FUNCTION_BLOCK FB_Depalletizer_1 IMPLEMENTS ITF_Depalletizer
VAR_INPUT
	Schuif : ITF_MotorSchuif;
	Zuignap1 : ITF_Vacuumzuignap;
	Zuignap2 : ITF_Vacuumzuignap;
	Zuignap3 : ITF_Vacuumzuignap;
	Zuignap4 : ITF_Vacuumzuignap;
	Druksensor1 : ITF_Druksensor;
	KlepDepallet : ITF_UnitKlep;

END_VAR
VAR_OUTPUT
END_VAR
VAR
	InputStateDep : E_PackMLStates;	
	CurrentStateDep : E_PackMLStates;



	testbool : BOOL;
	testbool2 : BOOL;
	GelezenStatusMotorSchuif : E_MotorSchuifStatus;
	GelezenStatusVacuumzuignap : E_VacuumzuignapStatus;
	GelezenDruk : REAL;
	GelezenStatusDruksensor : E_DruksensorStatus;
END_VAR

CASE InputStateDep OF

    E_PackMLStates.Idle:
        Idle();

    E_PackMLStates.Starting:
        Starting();

    E_PackMLStates.Execute:
        Execute();

    E_PackMLStates.Resetting:
        Resetting();

    E_PackMLStates.Holding:
        Holding();

    E_PackMLStates.Held:
        Held();

    E_PackMLStates.Unholding:
        Unholding();

    E_PackMLStates.Suspending:
        Suspending();

    E_PackMLStates.Suspended:
        Suspended();

    E_PackMLStates.Unsuspending:
        Unsuspending();

    E_PackMLStates.Stopping:
        Stopping();

    E_PackMLStates.Stopped:
        Stopped();

    E_PackMLStates.Aborting:
        Aborting();

    E_PackMLStates.Aborted:
        Aborted();

    E_PackMLStates.Clearing:
        Clearing();

END_CASE


















IF testbool = TRUE THEN
	Schuif.SturingKort();
	Zuignap1.Loslaten();
END_IF

IF testbool2 = TRUE THEN
	Schuif.SturingLang();
	Zuignap1.Oppakken();
END_IF

GelezenStatusMotorSchuif := Schuif.Status;
GelezenStatusVacuumzuignap := Zuignap1.Status;
GelezenDruk := Druksensor1.Druk;
GelezenStatusDruksensor := Druksensor1.Status;

METHOD Aborted : BOOL
VAR_INPUT
END_VAR
END_METHOD

METHOD Aborting : BOOL
VAR_INPUT
END_VAR
END_METHOD

METHOD Clearing : BOOL
VAR_INPUT
END_VAR
END_METHOD

PROPERTY CurrentState : E_PackMLStates
GET
CurrentState := CurrentStateDep;
END_GET
SET
CurrentStateDep := CurrentState;
END_SET
END_PROPERTY

METHOD Execute : BOOL
VAR_INPUT
END_VAR
END_METHOD

METHOD Held : BOOL
VAR_INPUT
END_VAR
END_METHOD

METHOD Holding : BOOL
VAR_INPUT
END_VAR
END_METHOD

METHOD Idle : BOOL
VAR_INPUT
END_VAR
CurrentStateDep := E_PackMLStates.Idle;
END_METHOD

PROPERTY InputState : E_PackMLStates
GET
InputState := InputStateDep;
END_GET
SET
InputStateDep := InputState;
END_SET
END_PROPERTY

METHOD Resetting : BOOL
VAR_INPUT
END_VAR
END_METHOD

METHOD Starting : BOOL
VAR_INPUT
END_VAR
CurrentStateDep := E_PackMLStates.Starting;

IF  Schuif.Status = E_MotorSchuifStatus.Kort AND Zuignap1.Status = E_VacuumzuignapStatus.SturingVacuumLoslaten AND
	Zuignap2.Status = E_VacuumzuignapStatus.SturingVacuumLoslaten AND Zuignap3.Status = E_VacuumzuignapStatus.SturingVacuumLoslaten AND
	Zuignap4.Status = E_VacuumzuignapStatus.SturingVacuumLoslaten AND DrukSensor1.Status = E_DruksensorStatus.SensorInputOk AND 
	KlepDepallet.Status = FALSE  THEN //vergeet de andere voorwaarden niet !!!!!
	
	CurrentStateDep := E_PackMLStates.Idle;
	ELSE
		Schuif.SturingKort();
		Zuignap1.Loslaten();
		Zuignap2.Loslaten();
		Zuignap3.Loslaten();
		Zuignap4.Loslaten();
		KlepDepallet.SturingOpen(FALSE); 
END_IF
END_METHOD

METHOD Stopped : BOOL
VAR_INPUT
END_VAR
END_METHOD

METHOD Stopping : BOOL
VAR_INPUT
END_VAR
END_METHOD

METHOD Suspended : BOOL
VAR_INPUT
END_VAR
END_METHOD

METHOD Suspending : BOOL
VAR_INPUT
END_VAR
END_METHOD

METHOD Unholding : BOOL
VAR_INPUT
END_VAR
END_METHOD

METHOD Unsuspending : BOOL
VAR_INPUT
END_VAR
END_METHOD

END_FUNCTION_BLOCK

(* stored: Version 1.1.0.1
   POU FB_Depalletizer_1: Id {604c825a-b299-42a4-9d94-06f2cd7a73fd}, SpecialFunc None
   Folder Methods: Id {41eb30da-c817-4a57-90b2-9b373696aeab}
   Folder Properties: Id {0a932fc3-77da-47ab-9595-fa212dce3ce7}
   Method Aborted: Id {0bfc1c67-cbbf-4ee0-9411-dfa1daf9e1fa}
   Method Aborting: Id {874fcde3-a461-43b7-8542-2e8c8f07c54a}
   Method Clearing: Id {a7e21cb3-b81b-4227-8a32-6a19ec30fdab}
   Property CurrentState: Id {5521c871-13ed-4e4c-a9b3-60eda6f215d2}
   Get Get: Id {abf65026-5da4-4773-9ad7-0771ec9a23a9}
   Set Set: Id {6aece2b5-c6a5-460d-8bf7-a59f80b5ecaa}
   Method Execute: Id {7bc828e8-56fb-4ceb-956d-11c06042b4fa}
   Method Held: Id {abf5bffe-4e53-4e4f-a0f2-17eb456b0638}
   Method Holding: Id {9ee0f93f-9ee6-40ae-91af-7b218154d752}
   Method Idle: Id {53c5baf1-bd08-4e97-999e-1b6af5cbd2b8}
   Property InputState: Id {4302f528-8764-4bef-8b72-acc9ee6f8e24}
   Get Get: Id {e211b0f1-ab3b-4059-8fd8-0ad7c175cd84}
   Set Set: Id {9bfc232a-27d2-4dce-a92e-4c3226aac6cf}
   Method Resetting: Id {86e32daa-1809-4afe-ae0a-050d304e9de2}
   Method Starting: Id {0c8238a0-26f8-4256-bb0d-748493f97bd5}
   Method Stopped: Id {862a4bb4-364c-4936-8d10-c75d515773a0}
   Method Stopping: Id {c84b4a38-09b8-40eb-889d-b8cb17a1f62f}
   Method Suspended: Id {10bd4b16-4905-4f00-a760-dfd80c61558a}
   Method Suspending: Id {6449bf5c-880a-49ff-a3c3-47582521d253}
   Method Unholding: Id {cdd257db-9d5b-420e-8b45-aa519fc7f0c5}
   Method Unsuspending: Id {d115c6be-b751-498a-bb2d-3f6dd5c17c4d} *)
